PROGRAM Motion

VAR
	
		

	X: FBMotion;
	Y: FBMotion;  
	AxisRefX: AXIS_REF;
	AxisRefY: AXIS_REF;
	ManualMove: BOOL;
	rTarget_Y: LREAL;
	rTarget_X: LREAL;
	PowerOffStop: BOOL;
	PowerOn: BOOL;
	Reset_X: BOOL;
	Reset_Y: BOOL;
	FindHome: BOOL;
	ManualSlotMove: BOOL;
	SlotVariableY: INT;
	SlotVariableX: INT;
	fbLifter: FB_Lifter;
	Nosto: BOOL;
	Lasku: BOOL;
	eMode: E_Mode := E_MODE.manual;
	eState: E_State;
	AutoInit: BOOL := FALSE;
	tonNostonLaskuDelay: TON := (PT := TIME#1s0ms);
	tonNostonNostoDelay: TON := (PT := TIME#1S0MS);
	tonLaskunLaskuDelay: TON := (PT:= TIME#1S0MS);
	tonXDelayEnnenYP2P: TON := (PT:= TIME#100MS);
	DelayStartNostonLasku: BOOL;
	DelayStartNostonNosto: BOOL;
	DelayStartLaskunLasku: BOOL;
	DelayStartXDelayEnnenYP2P: BOOL;
END_VAR

//X-akseli
X(AxisRef:= AxisRefX, bHomeCalibrationCam:=(IO.Anturi_X_1));

//Y-akseli
Y(AxisRef:= AxisRefY, bHomeCalibrationCam:=(IO.Anturi_Y_3));

//fbLifter();
//IO.bLifter := fbLifter.bLifter;
//IO.Imukuppi := fbLifter.bImukuppi;

tonNostonLaskuDelay(IN:= DelayStartNostonLasku);
tonNostonNostoDelay(IN:= DelayStartNostonNosto);
tonLaskunLaskuDelay(IN:= DelayStartLaskunLasku);
tonXDelayEnnenYP2P(IN:= DelayStartXDelayEnnenYP2P);

CASE eMode OF
	E_Mode.manual:		
		IF ManualMove THEN
			Y.P2P(rTarget_Y);
			X.P2P(rTarget_X);
			ManualMove := FALSE;
		END_IF
		
		IF ManualSlotMove THEN
			Y.P2P(Slots.Coords[SlotVariableY].y);
			X.P2P(Slots.Coords[SlotVariableX].x);
			ManualSlotMove := FALSE;
		END_IF
		
		IF Reset_X THEN
			X.Reset();
			Reset_X := FALSE;
		END_IF
		
		IF Reset_Y THEN
			Y.Reset();
			Reset_Y := FALSE;
		END_IF
		
		
		IF PowerOffStop THEN
			X.PowerOff();
			Y.PowerOff();
			PowerOffStop := FALSE;
		END_IF
		
		IF PowerOn THEN
			X.PowerOn();
			Y.PowerOn();
			PowerOn := FALSE;
		END_IF
		
		IF FindHome THEN
			X.FindHome();
			IF X.bHomed THEN
				Y.FindHome();
				FindHome := FALSE;
			END_IF
			
		END_IF
		
		IF Nosto THEN
			fbLifter.KplNosto();
			Nosto := FALSE;
		END_IF
		
		IF Lasku THEN
			fbLifter.KplLasku();
			Lasku := FALSE;
		END_IF
	
	E_Mode.auto:
		CASE eState OF
			E_State.inactive:
				IF AutoInit THEN
					AutoInit:= FALSE;
					X.PowerOn();
					Y.PowerOn();
					eState := E_state.initialising;
				END_IF
	
			E_State.initialising:
				IF X.bPowerStatus AND Y.bPowerStatus THEN
					X.FindHome();
					//Y.FindHome();
					eState := E_state.homing;
				END_IF
			
			E_State.homing:
				IF X.bHomed  THEN //AND Y.bHomed THEN
					Y.FindHome();		
					IF Y.bHomed THEN
						eState := E_state.ready;	
					END_IF		
				END_IF
				
			E_State.ready:
				IF Comms.bSlotCmd THEN
					Comms.bSlotCmd := FALSE;
					X.P2P(Slots.Coords[Comms.stSlotCmd.from_slot].x);
					Y.P2P(Slots.Coords[Comms.stSlotCmd.from_slot].y);
					eState := E_state.move2pick;
				ELSIF Comms.kotiutusnappi THEN
					Comms.kotiutusnappi := FALSE;
					Y.P2P(0.0);
					X.P2P(0.0);
					eState := E_state.kotiutusnappi;
				END_IF
				
			E_State.move2pick:
				IF X.bP2P_Ready AND Y.bP2P_Ready THEN
					// fbLifter.KplNosto();
					IO.Nostin := TRUE;
					tonNostonLaskuDelay.PT := T#1S;
					DelayStartNostonLasku := TRUE;
					IF tonNostonLaskuDelay.Q THEN
						DelayStartNostonLasku := FALSE;
						Y.P2P(AxisRefY.NcToPlc.ActPos + 100);
						eState := E_state.pick;
					END_IF
				END_IF
				
			E_State.pick:
				IF Y.bP2P_Ready THEN
					IO.Nostin := FALSE;
					tonNostonNostoDelay.PT := T#1S;
					DelayStartNostonNosto := TRUE;
					IF tonNostonNostoDelay.Q THEN
						DelayStartNostonNosto := FALSE;
						Y.P2P(AxisRefY.NcToPlc.ActPos - 100);
						eState := E_state.pick2;
					END_IF
				END_IF;
					
			E_State.pick2:
				IF Y.bP2P_Ready THEN
					X.P2P(Slots.Coords[Comms.stSlotCmd.to_slot].x);
					eState := E_state.pick3;
				END_IF
				
			E_State.pick3:
				IF X.bP2P_Ready THEN
					Y.P2P(Slots.Coords[Comms.stSlotCmd.to_slot].y + 100);
					eState := E_state.move2place;
				END_IF
				
			E_State.move2place:
				IF X.bP2P_Ready AND Y.bP2P_Ready THEN
					// fbLifter.KplLasku();
					IO.Nostin := TRUE;
					tonLaskunLaskuDelay.PT := T#1S;
					DelayStartLaskunLasku := TRUE;
					IF tonLaskunLaskuDelay.Q THEN
						DelayStartLaskunLasku := FALSE;
						Y.P2P(AxisRefY.NcToPlc.ActPos - 100);
						eState := E_state.place;
					END_IF
				END_IF
				
			E_State.place:
				IF X.bP2P_Ready AND Y.bP2P_Ready THEN
					IO.Nostin := FALSE;
					eState := E_state.ready;
				END_IF;

			E_State.kotiutusnappi:
				IF X.bP2P_Ready AND Y.bP2P_Ready THEN
					eState := E_state.ready;
				END_IF;
		END_CASE
END_CASE

END_PROGRAM

(* stored: Version 1.1.0.1, ProductVersion 3.1.4024.12
   POU Motion: Id {001a247c-a044-487c-a28e-44191cbf5c4a}, SpecialFunc None *)
